TYPE T_CASE_Barcode : T_MaxString;
END_TYPE

(* stored: Version 1.1.0.1, ProductVersion 3.1.4024.15
   DUT T_CASE_Barcode: Id {c04a7e7f-6b82-4879-b2b0-41cddfb41c8a} *)
